PROGRAM MAIN
VAR
	i_Result1 : RS232_Return;
	i_Result2 : RS232_Return;
	i_Result3 : RS232_Return;
END_VAR

i_Result1 := RS232(w_RS232Input:= 16#1D06);
i_Result2 := RS232(w_RS232Input:= 16#534C);
i_Result3 := RS232(w_RS232Input:= 16#C705);

END_PROGRAM

(* stored: Version 1.1.0.1, ProductVersion 3.1.4022.12
   POU MAIN: Id {bd44c13e-0269-4594-9737-df5f93033b95}, SpecialFunc None *)
